// SIMATIC S7-200 SMART project (STEP 7-Micro/WIN SMART), CPU CR40

ORGANIZATION_BLOCK MAIN:OB1
TITLE=程序注释
BEGIN
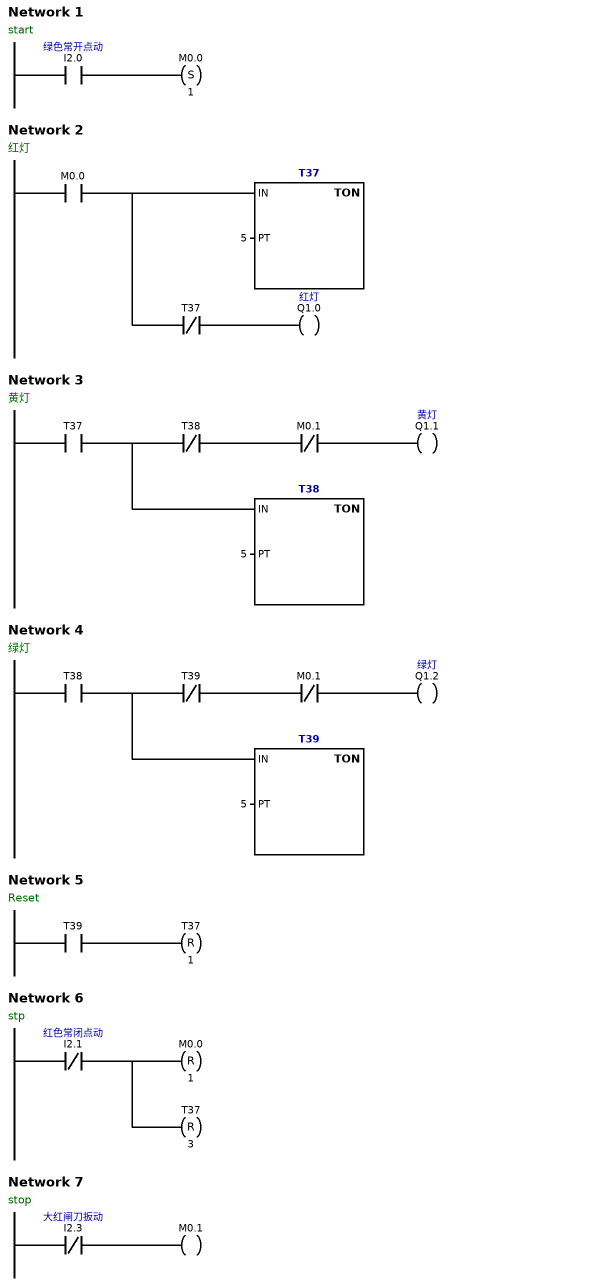
Network 1
// start
LD     绿色常开点动:I2.0
S      M0.0, 1
Network 2
// 红灯
LD     M0.0
TON    T37, 5
AN     T37
=      红灯:Q1.0
Network 3
// 黄灯
LD     T37
LPS
AN     T38
AN     M0.1
=      黄灯:Q1.1
LPP
TON    T38, 5
Network 4
// 绿灯
LD     T38
LPS
AN     T39
AN     M0.1
=      绿灯:Q1.2
LPP
TON    T39, 5
Network 5
// Reset
LD     T39
R      T37, 1
Network 6
// stp
LDN    红色常闭点动:I2.1
R      M0.0, 1
R      T37, 3
Network 7
// stop
LDN    大红闸刀扳动:I2.3
=      M0.1
END_ORGANIZATION_BLOCK
